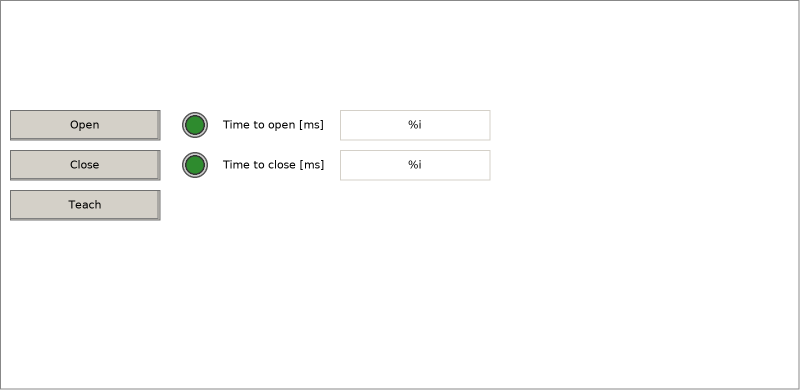
VISUALIZATION VisuCylinderControl  // 800x390
VAR_IN_OUT
	fbManualControler	: FB_ManualController ;
END_VAR
    Button (10,110 150x30), "Open"
        tap fbManualControler.pDevCylinder^.stManualCtrl.bCmdOpen
    Button (10,150 150x30), "Close"
        tap fbManualControler.pDevCylinder^.stManualCtrl.bCmdClose
    Lamp1 (180,110 30x30), variable: fbManualControler.pDevCylinder^.bFco_Open, style: Lamp-Lamp1-Green
    Button (10,190 150x30), "Teach"
        toggle fbManualControler.pDevCylinder^.stManualCtrl.bCmdTeach
    Lamp1 (180,150 30x30), variable: fbManualControler.pDevCylinder^.bFco_Closed, style: Lamp-Lamp1-Green
    Label (220,110 100x30), "Time to open [ms]"
    Label (220,150 100x30), "Time to close [ms]"
    Textfield (340,150 150x30), "%i", text variable: fbManualControler.pDevCylinder^.stParTimeToClose.fValue
        OnMouseClick: write the text variable via VisuDialogs.Numpad, min 0
    Textfield (340,110 150x30), "%i", text variable: fbManualControler.pDevCylinder^.stParTimeToOpen.fValue
        OnMouseClick: write the text variable via VisuDialogs.Numpad, min 0
END_VISUALIZATION

(* stored: Version 1.1.0.1, ProductVersion 3.1.4024.11
   Visu VisuCylinderControl: Id {094ca4d5-2080-09e7-2c82-cf5dd647e70f} *)
